// TIA Portal project "P4" (V17)

(* hardware
DEVICE "S7-1500/ET200MP station_1"  S7-1500 station
   slot 0: "Rail_0"  Rack  6ES7 590-1***0-0AA0
   slot 1: "PLC_1"  CPU 1515-2 PN  6ES7 515-2AM02-0AB0  V2.9
      slot 3: "CPU display_1"  6ES7591-1BA00-0AA0
      slot 32768: "PROFINET interface_1"  X1
         slot 32769: "Port_1"  X1 P1
         slot 32770: "Port_2"  X1 P2
      slot 33024: "PROFINET interface_2"  X2
         slot 33025: "Port_1"  X2 P1
      slot 34817: "Virtual CP interface port_1"  Virtual CP interface port  Virtual CP interface port
*)

// ===== PLC "PLC_1"  CPU 1515-2 PN =====

VAR_GLOBAL   // PLC tag table "Default tag table"
   "START PB" AT %E0.0 : Bool;
   "STOP PB" AT %E0.1 : Bool;
   "LS 1" AT %E0.2 : Bool;
   "LS 2" AT %E0.3 : Bool;
   "LS 3" AT %E0.4 : Bool;
   "LSDN" AT %E0.5 : Bool;
   "LSUP" AT %E0.6 : Bool;
   "RELAY COIL" AT %M0.0 : Bool;
   "RELAY COIL 1" AT %M0.1 : Bool;
   "RELAY COIL 2" AT %M0.2 : Bool;
   "RELAY COIL 3" AT %M0.3 : Bool;
   "RELAY COIL 4" AT %M0.4 : Bool;
   "UP_MOTOR" AT %A0.0 : Bool;
   "DN_MOTOR" AT %A0.1 : Bool;
   "CONVEYOR MOTOR" AT %A0.2 : Bool;
END_VAR

ORGANIZATION_BLOCK "Main"   // OB1, LAD, ProgramCycle
TITLE = "Main Program Sweep (Cycle)"
{ S7_Optimized_Access := 'TRUE' }
VERSION : 0.1
   VAR_INPUT
      Initial_Call : Bool;   // Initial call of this OB
      Remanence : Bool;   // =True, if remanent data are available
   END_VAR
BEGIN

REGION Network 1
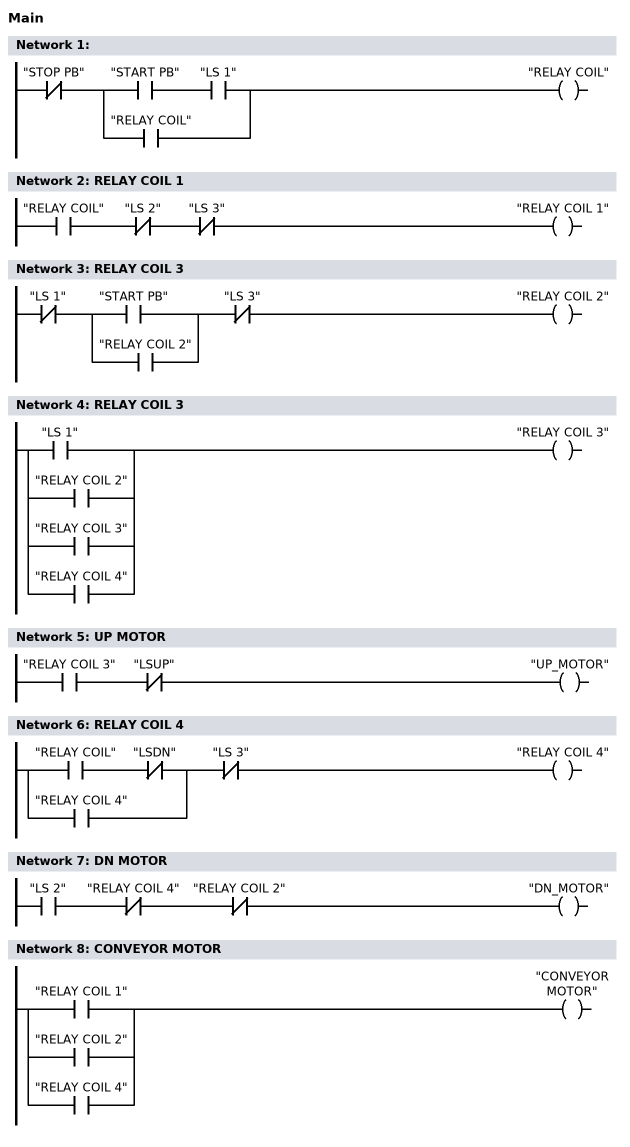
   RUNG wire#powerrail
      I_Contact( "STOP PB" )
      wire#w1
      Contact( "START PB" )
      Contact( "LS 1" )
      wire#w2
      Coil( "RELAY COIL" )
   END_RUNG
   RUNG wire#w1
      Contact( "RELAY COIL" )
   END_RUNG wire#w2
   // the same network as SCL:
   "RELAY COIL" := NOT "STOP PB" AND (("START PB" AND "LS 1") OR "RELAY COIL");
END_REGION

REGION Network 2: RELAY COIL 1
   RUNG wire#powerrail
      Contact( "RELAY COIL" )
      I_Contact( "LS 2" )
      I_Contact( "LS 3" )
      Coil( "RELAY COIL 1" )
   END_RUNG
   // the same network as SCL:
   "RELAY COIL 1" := "RELAY COIL" AND NOT "LS 2" AND NOT "LS 3";
END_REGION

REGION Network 3: RELAY COIL 3
   RUNG wire#powerrail
      I_Contact( "LS 1" )
      wire#w1
      Contact( "START PB" )
      wire#w2
      I_Contact( "LS 3" )
      Coil( "RELAY COIL 2" )
   END_RUNG
   RUNG wire#w1
      Contact( "RELAY COIL 2" )
   END_RUNG wire#w2
   // the same network as SCL:
   "RELAY COIL 2" := NOT "LS 1" AND ("START PB" OR "RELAY COIL 2") AND NOT "LS 3";
END_REGION

REGION Network 4: RELAY COIL 3
   RUNG wire#powerrail
      Contact( "LS 1" )
      wire#w1
      Coil( "RELAY COIL 3" )
   END_RUNG
   RUNG wire#powerrail
      Contact( "RELAY COIL 2" )
   END_RUNG wire#w1
   RUNG wire#powerrail
      Contact( "RELAY COIL 3" )
   END_RUNG wire#w1
   RUNG wire#powerrail
      Contact( "RELAY COIL 4" )
   END_RUNG wire#w1
   // the same network as SCL:
   "RELAY COIL 3" := "LS 1" OR "RELAY COIL 2" OR "RELAY COIL 3" OR "RELAY COIL 4";
END_REGION

REGION Network 5: UP MOTOR
   RUNG wire#powerrail
      Contact( "RELAY COIL 3" )
      I_Contact( "LSUP" )
      Coil( "UP_MOTOR" )
   END_RUNG
   // the same network as SCL:
   "UP_MOTOR" := "RELAY COIL 3" AND NOT "LSUP";
END_REGION

REGION Network 6: RELAY COIL 4
   RUNG wire#powerrail
      Contact( "RELAY COIL" )
      I_Contact( "LSDN" )
      wire#w1
      I_Contact( "LS 3" )
      Coil( "RELAY COIL 4" )
   END_RUNG
   RUNG wire#powerrail
      Contact( "RELAY COIL 4" )
   END_RUNG wire#w1
   // the same network as SCL:
   "RELAY COIL 4" := (("RELAY COIL" AND NOT "LSDN") OR "RELAY COIL 4") AND NOT "LS 3";
END_REGION

REGION Network 7: DN MOTOR
   RUNG wire#powerrail
      Contact( "LS 2" )
      I_Contact( "RELAY COIL 4" )
      I_Contact( "RELAY COIL 2" )
      Coil( "DN_MOTOR" )
   END_RUNG
   // the same network as SCL:
   "DN_MOTOR" := "LS 2" AND NOT "RELAY COIL 4" AND NOT "RELAY COIL 2";
END_REGION

REGION Network 8: CONVEYOR MOTOR
   RUNG wire#powerrail
      Contact( "RELAY COIL 1" )
      wire#w1
      Coil( "CONVEYOR MOTOR" )
   END_RUNG
   RUNG wire#powerrail
      Contact( "RELAY COIL 2" )
   END_RUNG wire#w1
   RUNG wire#powerrail
      Contact( "RELAY COIL 4" )
   END_RUNG wire#w1
   // the same network as SCL:
   "CONVEYOR MOTOR" := "RELAY COIL 1" OR "RELAY COIL 2" OR "RELAY COIL 4";
END_REGION
END_ORGANIZATION_BLOCK